PROGRAM MAIN
VAR
END_VAR

Prg_Loops();

END_PROGRAM

(* stored: Version 1.1.0.1, ProductVersion 3.1.4024.9
   POU MAIN: Id {5e7e705a-294f-4118-a5ed-89edb59061c5}, SpecialFunc None *)
